// TIA Portal V16 export
// export: Created 2025-08-01T13:37:56.5430103Z, ExportSetting WithDefaults, DisplayName Totally Integrated Automation Portal, DisplayVersion V16, DisplayName TIA Portal Version Control Interface, DisplayVersion V16, DisplayName TIA Portal Openness, DisplayVersion V16, DisplayName STEP 7 Professional, DisplayVersion V16, DisplayName STEP 7 Safety, DisplayVersion V16, DisplayName WinCC Advanced, DisplayVersion V16
FUNCTION "1 - Outputs" : Void   // FC5, LAD
VERSION : 0.1
// This Function program is for operating the machine automatic and manual.
// stored: AutoNumber true, IsIECCheckEnabled false, UDAEnableTagReadback false
   VAR_TEMP
      Valve_2_Pulse : Bool;
      BlowOff_Activated : Bool;
      BlowOffManual : Bool;
      Pulse1 : Bool;
      Drive_1_ReferenceRun : Bool;
   END_VAR
   VAR_TEMP   // added for the SCL form of the ladder/FBD networks
      _w1 : Bool;
   END_VAR
BEGIN

REGION Network 1: Drive 1 - Control
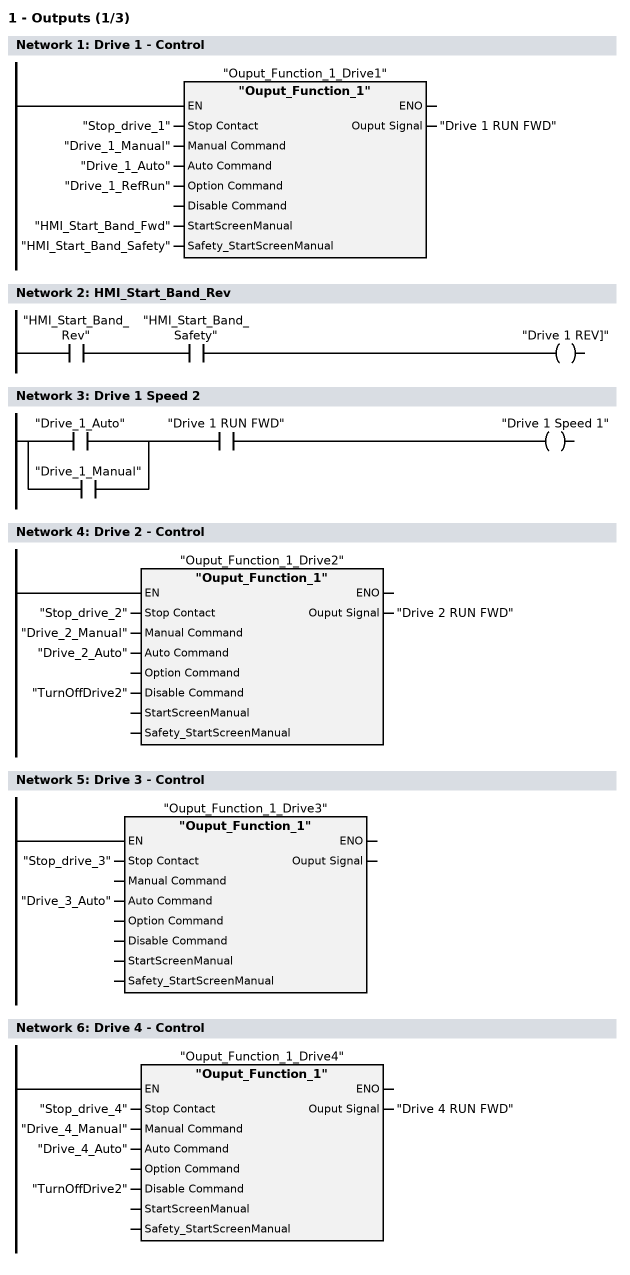
   RUNG wire#powerrail
      "Ouput_Function_1_Drive1"("Stop Contact" := "Stop_drive_1", "Manual Command" := "Drive_1_Manual", "Auto Command" := "Drive_1_Auto", "Option Command" := "Drive_1_RefRun", "Disable Command" :=, StartScreenManual := "HMI_Start_Band_Fwd", Safety_StartScreenManual := "HMI_Start_Band_Safety", "Ouput Signal" => "Drive 1 RUN FWD")
   END_RUNG
   // the same network as SCL:
   "Ouput_Function_1_Drive1"("Stop Contact" := "Stop_drive_1",   // "Ouput_Function_1"
                           "Manual Command" := "Drive_1_Manual",
                           "Auto Command" := "Drive_1_Auto",
                           "Option Command" := "Drive_1_RefRun",
                           StartScreenManual := "HMI_Start_Band_Fwd",
                           Safety_StartScreenManual := "HMI_Start_Band_Safety",
                           "Ouput Signal" => "Drive 1 RUN FWD");
END_REGION

REGION Network 2: HMI_Start_Band_Rev
   RUNG wire#powerrail
      Contact( "HMI_Start_Band_Rev" )
      Contact( "HMI_Start_Band_Safety" )
      Coil( "Drive 1 REV]" )
   END_RUNG
   // the same network as SCL:
   "Drive 1 REV]" := "HMI_Start_Band_Rev" AND "HMI_Start_Band_Safety";
END_REGION

REGION Network 3: Drive 1 Speed 2
   RUNG wire#powerrail
      Contact( "Drive_1_Auto" )
      wire#w1
      Contact( "Drive 1 RUN FWD" )
      Coil( "Drive 1 Speed 1" )
   END_RUNG
   RUNG wire#powerrail
      Contact( "Drive_1_Manual" )
   END_RUNG wire#w1
   // the same network as SCL:
   "Drive 1 Speed 1" := ("Drive_1_Auto" OR "Drive_1_Manual") AND "Drive 1 RUN FWD";
END_REGION

REGION Network 4: Drive 2 - Control
   RUNG wire#powerrail
      "Ouput_Function_1_Drive2"("Stop Contact" := "Stop_drive_2", "Manual Command" := "Drive_2_Manual", "Auto Command" := "Drive_2_Auto", "Option Command" :=, "Disable Command" := "TurnOffDrive2", StartScreenManual :=, Safety_StartScreenManual :=, "Ouput Signal" => "Drive 2 RUN FWD")
   END_RUNG
   // the same network as SCL:
   "Ouput_Function_1_Drive2"("Stop Contact" := "Stop_drive_2",   // "Ouput_Function_1"
                           "Manual Command" := "Drive_2_Manual",
                           "Auto Command" := "Drive_2_Auto",
                           "Disable Command" := "TurnOffDrive2",
                           "Ouput Signal" => "Drive 2 RUN FWD");
END_REGION

REGION Network 5: Drive 3 - Control
   RUNG wire#powerrail
      "Ouput_Function_1_Drive3"("Stop Contact" := "Stop_drive_3", "Manual Command" :=, "Auto Command" := "Drive_3_Auto", "Option Command" :=, "Disable Command" :=, StartScreenManual :=, Safety_StartScreenManual :=, "Ouput Signal" =>)
   END_RUNG
   // the same network as SCL:
   "Ouput_Function_1_Drive3"("Stop Contact" := "Stop_drive_3", "Auto Command" := "Drive_3_Auto");   // "Ouput_Function_1"
END_REGION

REGION Network 6: Drive 4 - Control
   RUNG wire#powerrail
      "Ouput_Function_1_Drive4"("Stop Contact" := "Stop_drive_4", "Manual Command" := "Drive_4_Manual", "Auto Command" := "Drive_4_Auto", "Option Command" :=, "Disable Command" := "TurnOffDrive2", StartScreenManual :=, Safety_StartScreenManual :=, "Ouput Signal" => "Drive 4 RUN FWD")
   END_RUNG
   // the same network as SCL:
   "Ouput_Function_1_Drive4"("Stop Contact" := "Stop_drive_4",   // "Ouput_Function_1"
                           "Manual Command" := "Drive_4_Manual",
                           "Auto Command" := "Drive_4_Auto",
                           "Disable Command" := "TurnOffDrive2",
                           "Ouput Signal" => "Drive 4 RUN FWD");
END_REGION

REGION Network 7: Drive 5 - Control
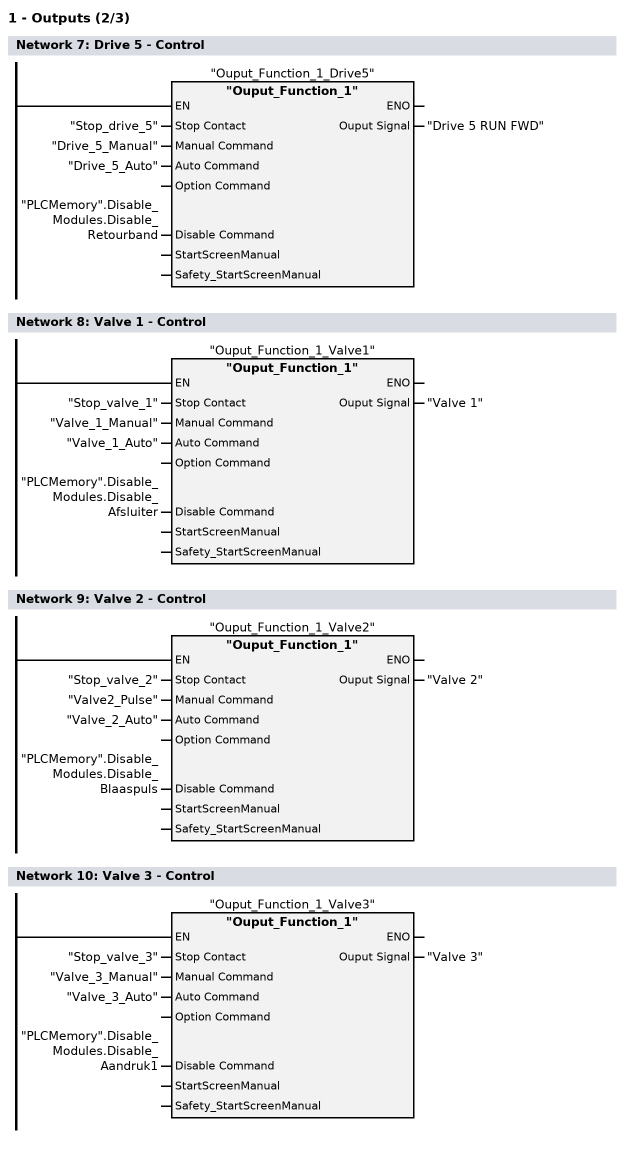
   RUNG wire#powerrail
      "Ouput_Function_1_Drive5"("Stop Contact" := "Stop_drive_5", "Manual Command" := "Drive_5_Manual", "Auto Command" := "Drive_5_Auto", "Option Command" :=, "Disable Command" := "PLCMemory".Disable_Modules.Disable_Retourband, StartScreenManual :=, Safety_StartScreenManual :=, "Ouput Signal" => "Drive 5 RUN FWD")
   END_RUNG
   // the same network as SCL:
   "Ouput_Function_1_Drive5"("Stop Contact" := "Stop_drive_5",   // "Ouput_Function_1"
                           "Manual Command" := "Drive_5_Manual",
                           "Auto Command" := "Drive_5_Auto",
                           "Disable Command" := "PLCMemory".Disable_Modules.Disable_Retourband,
                           "Ouput Signal" => "Drive 5 RUN FWD");
END_REGION

REGION Network 8: Valve 1 - Control
   RUNG wire#powerrail
      "Ouput_Function_1_Valve1"("Stop Contact" := "Stop_valve_1", "Manual Command" := "Valve_1_Manual", "Auto Command" := "Valve_1_Auto", "Option Command" :=, "Disable Command" := "PLCMemory".Disable_Modules.Disable_Afsluiter, StartScreenManual :=, Safety_StartScreenManual :=, "Ouput Signal" => "Valve 1")
   END_RUNG
   // the same network as SCL:
   "Ouput_Function_1_Valve1"("Stop Contact" := "Stop_valve_1",   // "Ouput_Function_1"
                           "Manual Command" := "Valve_1_Manual",
                           "Auto Command" := "Valve_1_Auto",
                           "Disable Command" := "PLCMemory".Disable_Modules.Disable_Afsluiter,
                           "Ouput Signal" => "Valve 1");
END_REGION

REGION Network 9: Valve 2 - Control
   RUNG wire#powerrail
      "Ouput_Function_1_Valve2"("Stop Contact" := "Stop_valve_2", "Manual Command" := "Valve2_Pulse", "Auto Command" := "Valve_2_Auto", "Option Command" :=, "Disable Command" := "PLCMemory".Disable_Modules.Disable_Blaaspuls, StartScreenManual :=, Safety_StartScreenManual :=, "Ouput Signal" => "Valve 2")
   END_RUNG
   // the same network as SCL:
   "Ouput_Function_1_Valve2"("Stop Contact" := "Stop_valve_2",   // "Ouput_Function_1"
                           "Manual Command" := "Valve2_Pulse",
                           "Auto Command" := "Valve_2_Auto",
                           "Disable Command" := "PLCMemory".Disable_Modules.Disable_Blaaspuls,
                           "Ouput Signal" => "Valve 2");
END_REGION

REGION Network 10: Valve 3 - Control
   RUNG wire#powerrail
      "Ouput_Function_1_Valve3"("Stop Contact" := "Stop_valve_3", "Manual Command" := "Valve_3_Manual", "Auto Command" := "Valve_3_Auto", "Option Command" :=, "Disable Command" := "PLCMemory".Disable_Modules.Disable_Aandruk1, StartScreenManual :=, Safety_StartScreenManual :=, "Ouput Signal" => "Valve 3")
   END_RUNG
   // the same network as SCL:
   "Ouput_Function_1_Valve3"("Stop Contact" := "Stop_valve_3",   // "Ouput_Function_1"
                           "Manual Command" := "Valve_3_Manual",
                           "Auto Command" := "Valve_3_Auto",
                           "Disable Command" := "PLCMemory".Disable_Modules.Disable_Aandruk1,
                           "Ouput Signal" => "Valve 3");
END_REGION

REGION Network 11: Valve 4 - Control
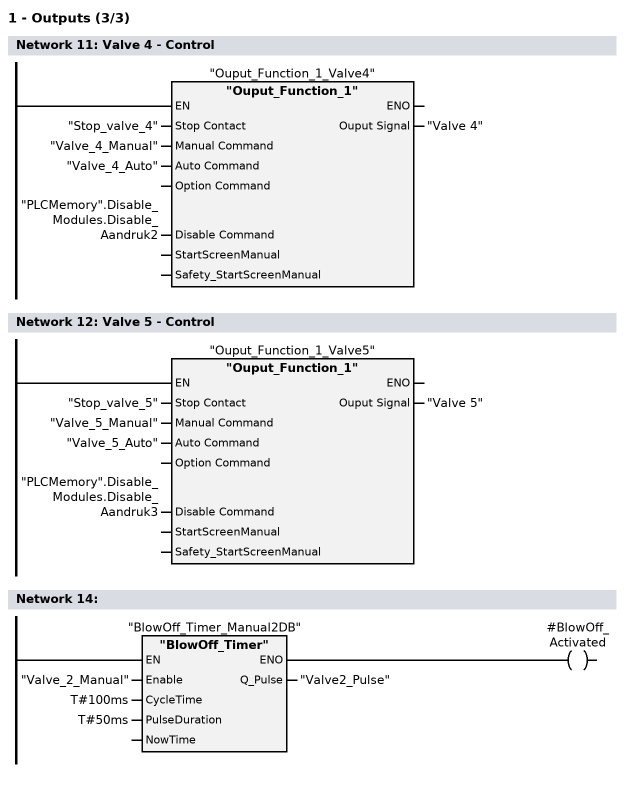
   RUNG wire#powerrail
      "Ouput_Function_1_Valve4"("Stop Contact" := "Stop_valve_4", "Manual Command" := "Valve_4_Manual", "Auto Command" := "Valve_4_Auto", "Option Command" :=, "Disable Command" := "PLCMemory".Disable_Modules.Disable_Aandruk2, StartScreenManual :=, Safety_StartScreenManual :=, "Ouput Signal" => "Valve 4")
   END_RUNG
   // the same network as SCL:
   "Ouput_Function_1_Valve4"("Stop Contact" := "Stop_valve_4",   // "Ouput_Function_1"
                           "Manual Command" := "Valve_4_Manual",
                           "Auto Command" := "Valve_4_Auto",
                           "Disable Command" := "PLCMemory".Disable_Modules.Disable_Aandruk2,
                           "Ouput Signal" => "Valve 4");
END_REGION

REGION Network 12: Valve 5 - Control
   RUNG wire#powerrail
      "Ouput_Function_1_Valve5"("Stop Contact" := "Stop_valve_5", "Manual Command" := "Valve_5_Manual", "Auto Command" := "Valve_5_Auto", "Option Command" :=, "Disable Command" := "PLCMemory".Disable_Modules.Disable_Aandruk3, StartScreenManual :=, Safety_StartScreenManual :=, "Ouput Signal" => "Valve 5")
   END_RUNG
   // the same network as SCL:
   "Ouput_Function_1_Valve5"("Stop Contact" := "Stop_valve_5",   // "Ouput_Function_1"
                           "Manual Command" := "Valve_5_Manual",
                           "Auto Command" := "Valve_5_Auto",
                           "Disable Command" := "PLCMemory".Disable_Modules.Disable_Aandruk3,
                           "Ouput Signal" => "Valve 5");
END_REGION

REGION Network 13: Blow Off Manual
END_REGION

REGION Network 14
   RUNG wire#powerrail
      "BlowOff_Timer_Manual2DB"(Enable := "Valve_2_Manual", CycleTime := T#100ms, PulseDuration := T#50ms, NowTime :=, Q_Pulse => "Valve2_Pulse")
      Coil( #BlowOff_Activated )
   END_RUNG
   // the same network as SCL:
   "BlowOff_Timer_Manual2DB"(Enable := "Valve_2_Manual",   // "BlowOff_Timer"
                           CycleTime := T#100ms,
                           PulseDuration := T#50ms,
                           Q_Pulse => "Valve2_Pulse",
                           ENO => #_w1);
   #BlowOff_Activated := #_w1;
END_REGION
END_FUNCTION
